% RSLogix 500 project P3_ABIOLA_A.RSS, saved by version 8.30.00.16 %
PROJECT "UNTITLED"    % processor: Bul.1763 MicroLogix 1100 Series B %

PROGRAM FILES
  LAD 2   2 rungs
  LAD 3 "PSEUDO IO"  30 rungs  % Contains all the assigned memery address used  %

DATA FILES
  O0 OUTPUT  4 elements
  I1 INPUT  6 elements
  S2 STATUS  66 elements
  B3 BINARY  1 elements
  T4 TIMER  7 elements
  C5 COUNTER  6 elements
  R6 CONTROL  1 elements
  N7 INTEGER  30 elements
  F8 FLOAT  1 elements
  ST9 STRFRBCSCN  50 elements  % Writes string from bar code scanner to PLC %

LADDER 2
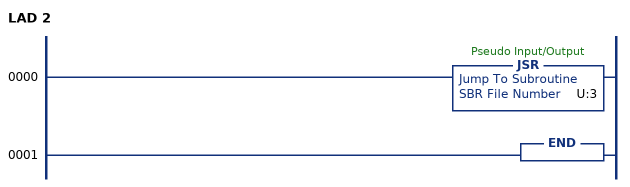
% Rung: 0 %
SOR JSR U:3 EOR
%   U:3  "Pseudo Input/Output" %
% Rung: 1 %
SOR END EOR

LADDER 3 "PSEUDO IO"    % Contains all the assigned memery address used  %
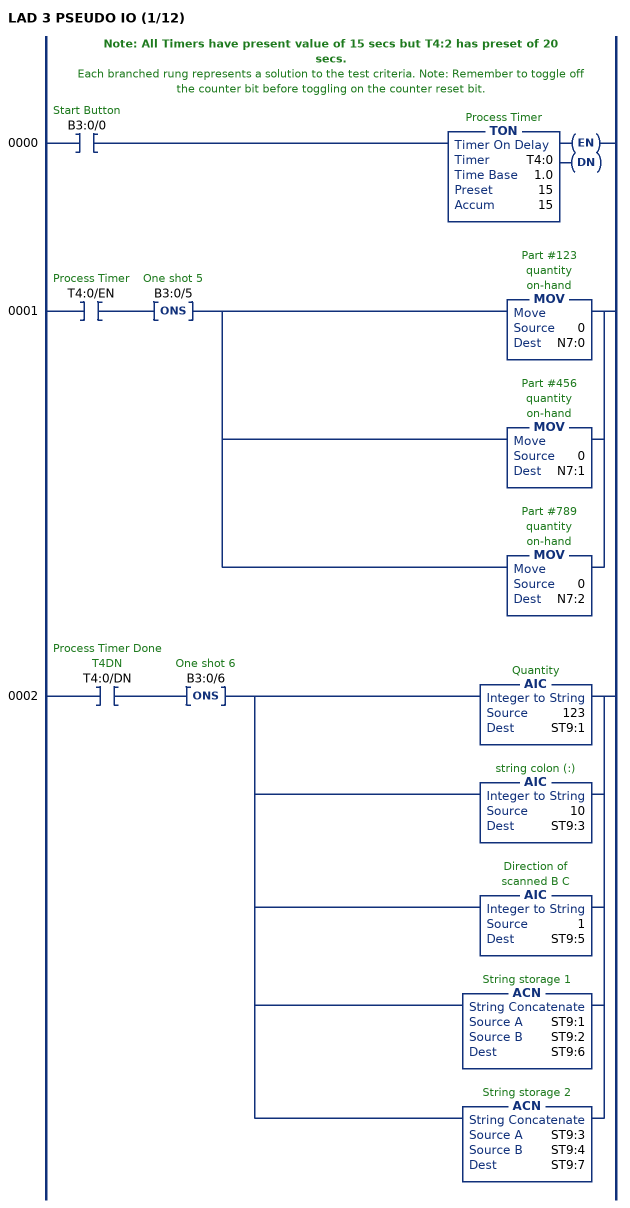
% Rung: 0 %
% TITLE: Note: All Timers have present value of 15 secs but T4:2 has preset of 20 secs. %
% Each branched rung represents a solution to the test criteria. Note: Remember to toggle off the counter bit before toggling on the counter reset bit. %
SOR XIC B3:0/0 TON T4:0 1.0 15 15 EOR
%   B3:0/0  "Start Button" %
%   T4:0  "Process Timer" %
% Rung: 1 %
SOR XIC T4:0/EN ONS B3:0/5 BST MOV 0 N7:0 NXB BST MOV 0 N7:1 NXB MOV 0 N7:2 BND BND EOR
%   T4:0  "Process Timer" %
%   B3:0/5  "One shot 5" %
%   N7:0  "Part #123 quantity on-hand" %
%   N7:1  "Part #456 quantity on-hand" %
%   N7:2  "Part #789 quantity on-hand" %
% Rung: 2 %
SOR XIC T4:0/DN ONS B3:0/6 BST AIC 123 ST9:1 NXB BST AIC 10 ST9:3 NXB BST AIC 1 ST9:5 NXB BST ACN ST9:1 ST9:2 ST9:6 NXB ACN ST9:3 ST9:4 ST9:7 BND BND BND BND EOR
%   T4:0/DN  T4DN  "Process Timer Done" %
%   B3:0/6  "One shot 6" %
%   ST9:1  "Quantity" %
%   ST9:3  "string colon (:)" %
%   ST9:5  "Direction of scanned B C" %
%   ST9:2  "String Quantity from Bar-code scanner" %
%   ST9:6  "String storage 1" %
%   ST9:4  "Concatination of colon (:) with direction from BCS" %
%   ST9:7  "String storage 2" %

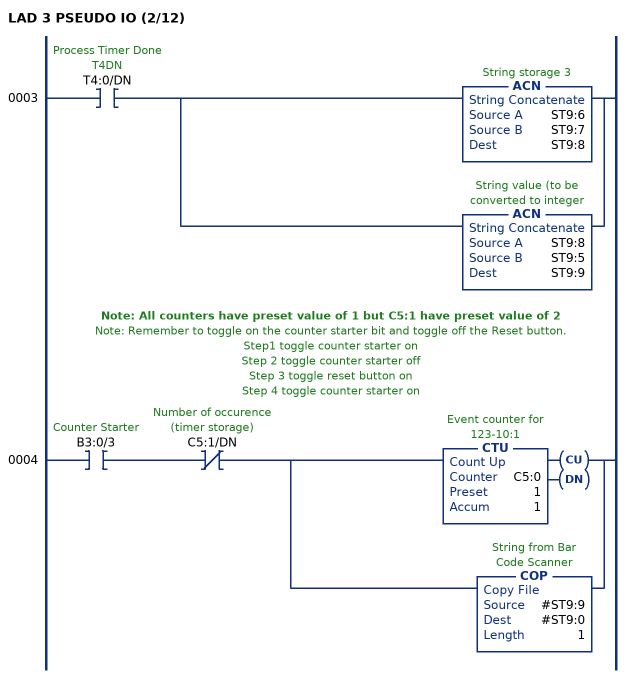
% Rung: 3 %
SOR XIC T4:0/DN BST ACN ST9:6 ST9:7 ST9:8 NXB ACN ST9:8 ST9:5 ST9:9 BND EOR
%   T4:0/DN  T4DN  "Process Timer Done" %
%   ST9:6  "String storage 1" %
%   ST9:7  "String storage 2" %
%   ST9:8  "String storage 3" %
%   ST9:5  "Direction of scanned B C" %
%   ST9:9  "String value (to be converted to integer" %
% Rung: 4 %
% TITLE: Note: All counters have preset value of 1 but C5:1 have preset value of 2 %
% Note: Remember to toggle on the counter starter bit and toggle off the Reset button.
% Step1 toggle counter starter on
% Step 2 toggle counter starter off
% Step 3 toggle reset button on
% Step 4 toggle counter starter on %
SOR XIC B3:0/3 XIO C5:1/DN BST CTU C5:0 1 1 NXB COP #ST9:9 #ST9:0 1 BND EOR
%   B3:0/3  "Counter Starter" %
%   C5:1/DN  "Number of occurence (timer storage)" %
%   C5:0  "Event counter for 123-10:1" %
%   ST9:9  "String value (to be converted to integer" %
%   ST9:0  "String from Bar Code Scanner" %

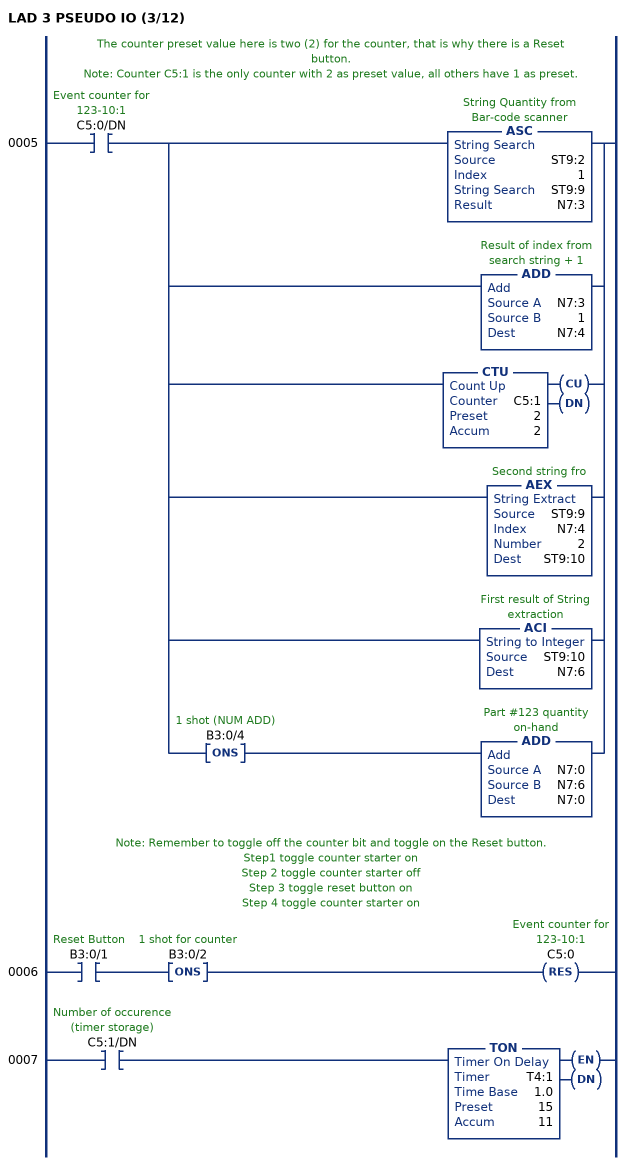
% Rung: 5 %
% The counter preset value here is two (2) for the counter, that is why there is a Reset button.
% Note: Counter C5:1 is the only counter with 2 as preset value, all others have 1 as preset. %
SOR XIC C5:0/DN BST BST ASC ST9:2 1 ST9:9 N7:3 NXB BST ADD N7:3 1 N7:4 NXB CTU C5:1 2 2 BND BND NXB BST AEX ST9:9 N7:4 2 ST9:10 NXB BST ACI ST9:10 N7:6 NXB ONS B3:0/4 ADD N7:0 N7:6 N7:0 BND BND BND EOR
%   C5:0  "Event counter for 123-10:1" %
%   ST9:2  "String Quantity from Bar-code scanner" %
%   ST9:9  "String value (to be converted to integer" %
%   N7:3  "Constant value of 10" %
%   N7:4  "Result of index from search string + 1" %
%   ST9:10  "Second string fro" %
%   N7:6  "First result of String extraction" %
%   B3:0/4  "1 shot (NUM ADD)" %
%   N7:0  "Part #123 quantity on-hand" %
% Rung: 6 %
% Note: Remember to toggle off the counter bit and toggle on the Reset button.
% Step1 toggle counter starter on
% Step 2 toggle counter starter off
% Step 3 toggle reset button on
% Step 4 toggle counter starter on %
SOR XIC B3:0/1 ONS B3:0/2 RES C5:0 EOR
%   B3:0/1  "Reset Button" %
%   B3:0/2  "1 shot for counter" %
%   C5:0  "Event counter for 123-10:1" %
% Rung: 7 %
SOR XIC C5:1/DN TON T4:1 1.0 15 11 EOR
%   C5:1/DN  "Number of occurence (timer storage)" %

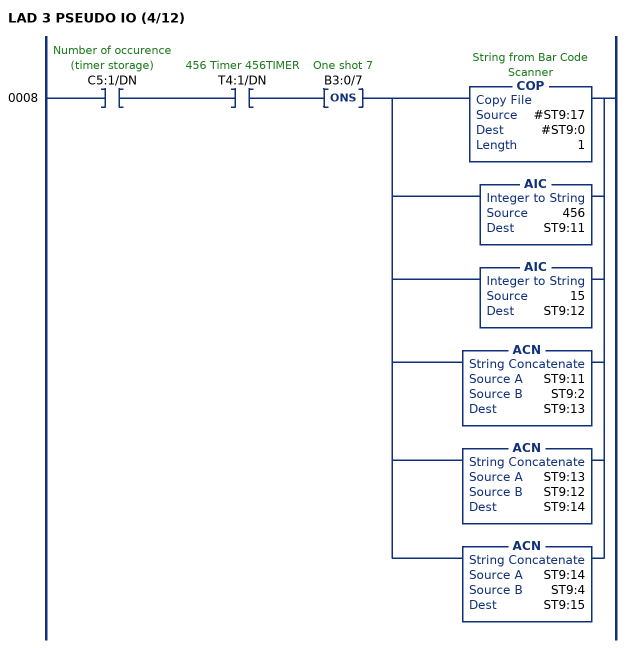
% Rung: 8 %
SOR XIC C5:1/DN XIC T4:1/DN ONS B3:0/7 BST BST COP #ST9:17 #ST9:0 1 NXB AIC 456 ST9:11 BND NXB AIC 15 ST9:12 NXB ACN ST9:11 ST9:2 ST9:13 NXB ACN ST9:13 ST9:12 ST9:14 NXB ACN ST9:14 ST9:4 ST9:15 BND EOR
%   C5:1/DN  "Number of occurence (timer storage)" %
%   T4:1/DN  456TIMER  "456 Timer" %
%   B3:0/7  "One shot 7" %
%   ST9:0  "String from Bar Code Scanner" %
%   ST9:2  "String Quantity from Bar-code scanner" %
%   ST9:4  "Concatination of colon (:) with direction from BCS" %

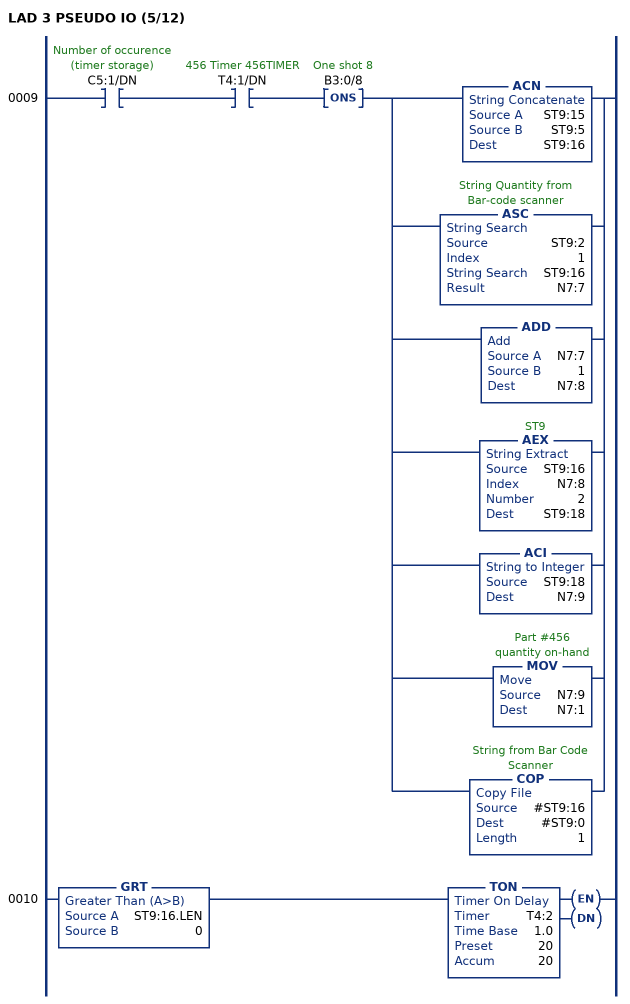
% Rung: 9 %
SOR XIC C5:1/DN XIC T4:1/DN ONS B3:0/8 BST ACN ST9:15 ST9:5 ST9:16 NXB ASC ST9:2 1 ST9:16 N7:7 NXB BST ADD N7:7 1 N7:8 NXB BST BST AEX ST9:16 N7:8 2 ST9:18 NXB ACI ST9:18 N7:9 BND NXB BST MOV N7:9 N7:1 NXB COP #ST9:16 #ST9:0 1 BND BND BND BND EOR
%   C5:1/DN  "Number of occurence (timer storage)" %
%   T4:1/DN  456TIMER  "456 Timer" %
%   B3:0/8  "One shot 8" %
%   ST9:5  "Direction of scanned B C" %
%   ST9:2  "String Quantity from Bar-code scanner" %
%   ST9:18  ST9 %
%   N7:1  "Part #456 quantity on-hand" %
%   ST9:0  "String from Bar Code Scanner" %
% Rung: 10 %
SOR GRT ST9:16.LEN 0 TON T4:2 1.0 20 20 EOR

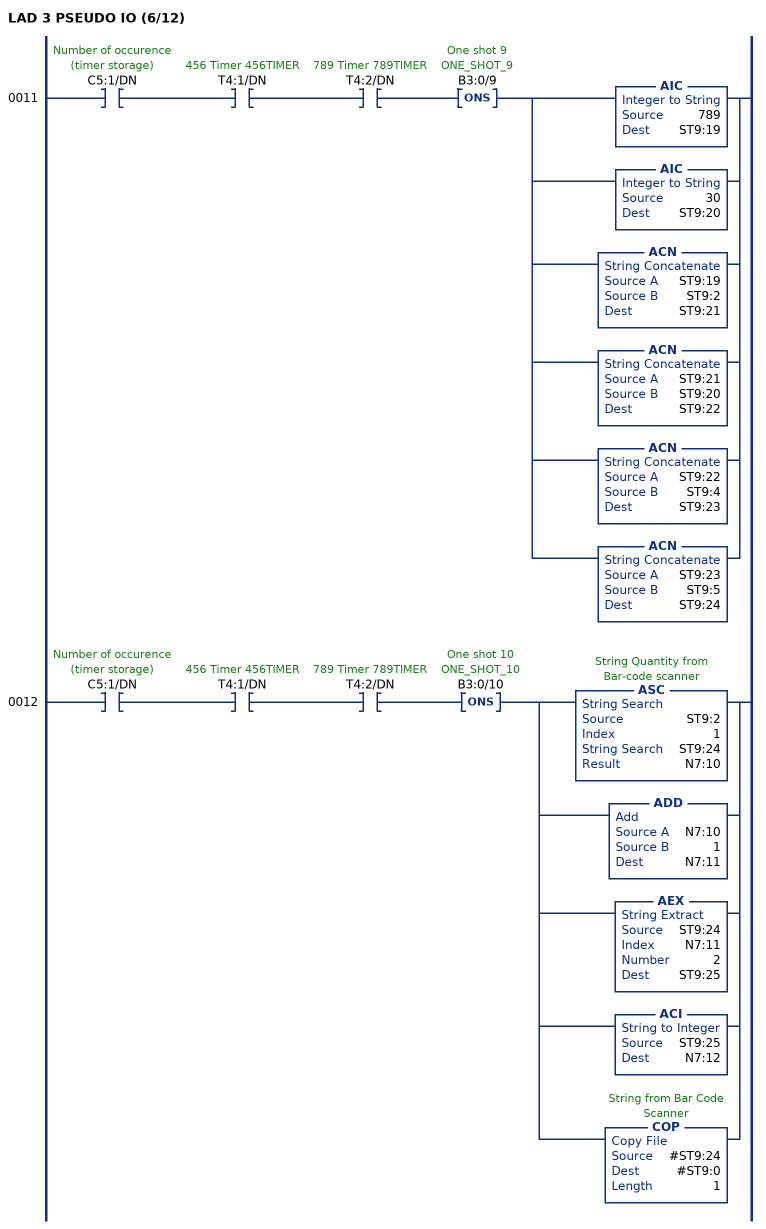
% Rung: 11 %
SOR XIC C5:1/DN XIC T4:1/DN XIC T4:2/DN ONS B3:0/9 BST AIC 789 ST9:19 NXB AIC 30 ST9:20 NXB ACN ST9:19 ST9:2 ST9:21 NXB ACN ST9:21 ST9:20 ST9:22 NXB ACN ST9:22 ST9:4 ST9:23 NXB ACN ST9:23 ST9:5 ST9:24 BND EOR
%   C5:1/DN  "Number of occurence (timer storage)" %
%   T4:1/DN  456TIMER  "456 Timer" %
%   T4:2/DN  789TIMER  "789 Timer" %
%   B3:0/9  ONE_SHOT_9  "One shot 9" %
%   ST9:2  "String Quantity from Bar-code scanner" %
%   ST9:4  "Concatination of colon (:) with direction from BCS" %
%   ST9:5  "Direction of scanned B C" %
% Rung: 12 %
SOR XIC C5:1/DN XIC T4:1/DN XIC T4:2/DN ONS B3:0/10 BST ASC ST9:2 1 ST9:24 N7:10 NXB BST ADD N7:10 1 N7:11 NXB BST AEX ST9:24 N7:11 2 ST9:25 NXB BST ACI ST9:25 N7:12 NXB COP #ST9:24 #ST9:0 1 BND BND BND BND EOR
%   C5:1/DN  "Number of occurence (timer storage)" %
%   T4:1/DN  456TIMER  "456 Timer" %
%   T4:2/DN  789TIMER  "789 Timer" %
%   B3:0/10  ONE_SHOT_10  "One shot 10" %
%   ST9:2  "String Quantity from Bar-code scanner" %
%   ST9:0  "String from Bar Code Scanner" %

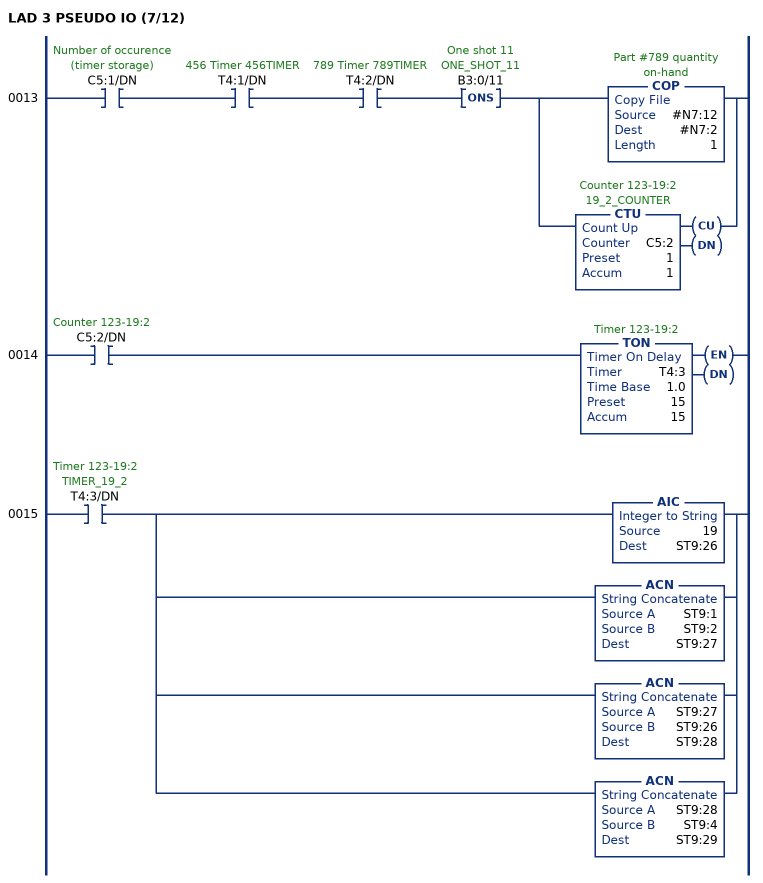
% Rung: 13 %
SOR XIC C5:1/DN XIC T4:1/DN XIC T4:2/DN ONS B3:0/11 BST COP #N7:12 #N7:2 1 NXB CTU C5:2 1 1 BND EOR
%   C5:1/DN  "Number of occurence (timer storage)" %
%   T4:1/DN  456TIMER  "456 Timer" %
%   T4:2/DN  789TIMER  "789 Timer" %
%   B3:0/11  ONE_SHOT_11  "One shot 11" %
%   N7:2  "Part #789 quantity on-hand" %
%   C5:2  19_2_COUNTER  "Counter 123-19:2" %
% Rung: 14 %
SOR XIC C5:2/DN TON T4:3 1.0 15 15 EOR
%   C5:2/DN  "Counter 123-19:2" %
%   T4:3  "Timer 123-19:2" %
% Rung: 15 %
SOR XIC T4:3/DN BST AIC 19 ST9:26 NXB BST ACN ST9:1 ST9:2 ST9:27 NXB BST ACN ST9:27 ST9:26 ST9:28 NXB ACN ST9:28 ST9:4 ST9:29 BND BND BND EOR
%   T4:3/DN  TIMER_19_2  "Timer 123-19:2" %
%   ST9:1  "Quantity" %
%   ST9:2  "String Quantity from Bar-code scanner" %
%   ST9:4  "Concatination of colon (:) with direction from BCS" %

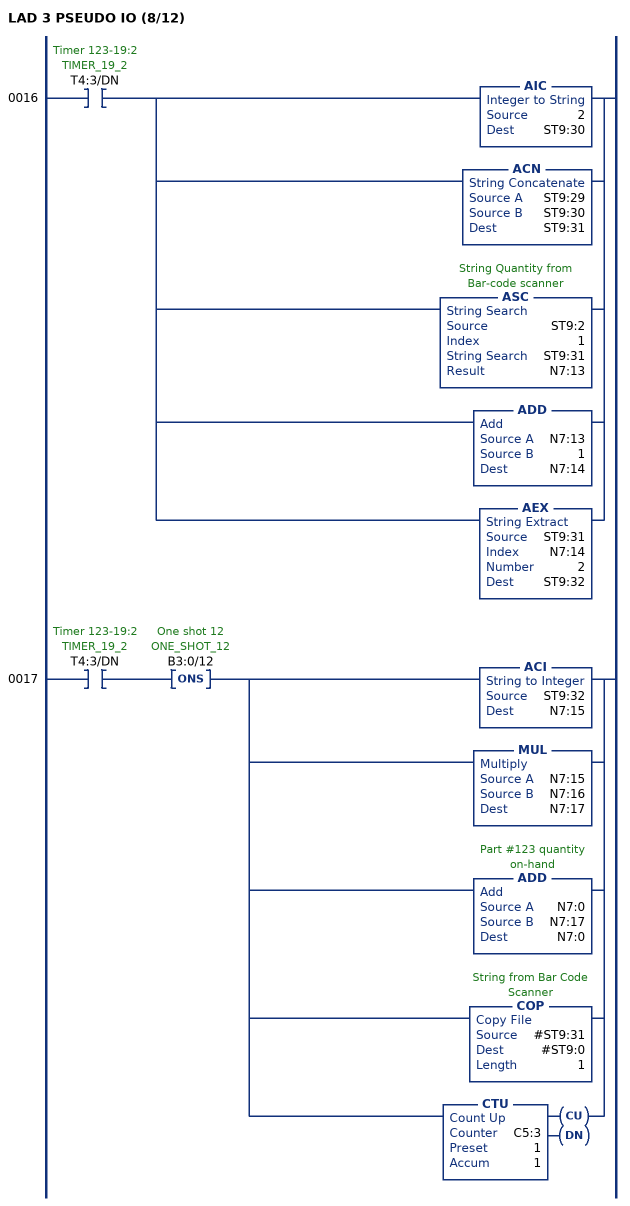
% Rung: 16 %
SOR XIC T4:3/DN BST AIC 2 ST9:30 NXB BST ACN ST9:29 ST9:30 ST9:31 NXB BST ASC ST9:2 1 ST9:31 N7:13 NXB BST ADD N7:13 1 N7:14 NXB AEX ST9:31 N7:14 2 ST9:32 BND BND BND BND EOR
%   T4:3/DN  TIMER_19_2  "Timer 123-19:2" %
%   ST9:2  "String Quantity from Bar-code scanner" %
% Rung: 17 %
SOR XIC T4:3/DN ONS B3:0/12 BST BST ACI ST9:32 N7:15 NXB MUL N7:15 N7:16 N7:17 BND NXB BST ADD N7:0 N7:17 N7:0 NXB BST COP #ST9:31 #ST9:0 1 NXB CTU C5:3 1 1 BND BND BND EOR
%   T4:3/DN  TIMER_19_2  "Timer 123-19:2" %
%   B3:0/12  ONE_SHOT_12  "One shot 12" %
%   N7:16  N %
%   N7:0  "Part #123 quantity on-hand" %
%   ST9:0  "String from Bar Code Scanner" %

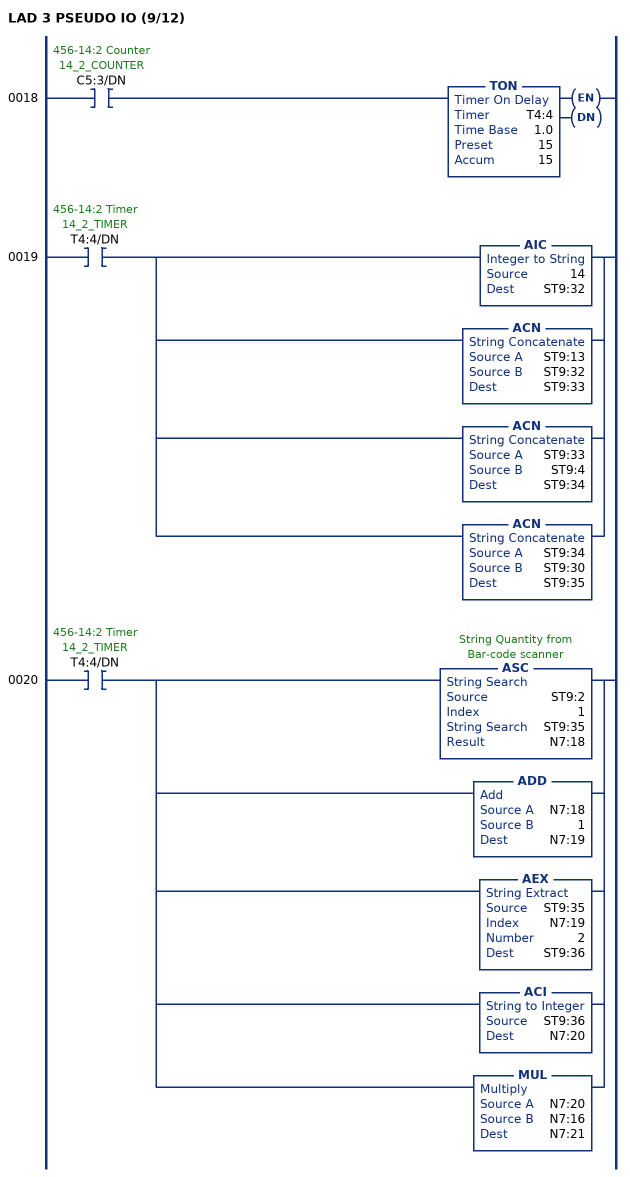
% Rung: 18 %
SOR XIC C5:3/DN TON T4:4 1.0 15 15 EOR
%   C5:3/DN  14_2_COUNTER  "456-14:2 Counter" %
% Rung: 19 %
SOR XIC T4:4/DN BST AIC 14 ST9:32 NXB BST ACN ST9:13 ST9:32 ST9:33 NXB BST ACN ST9:33 ST9:4 ST9:34 NXB ACN ST9:34 ST9:30 ST9:35 BND BND BND EOR
%   T4:4/DN  14_2_TIMER  "456-14:2 Timer" %
%   ST9:4  "Concatination of colon (:) with direction from BCS" %
% Rung: 20 %
SOR XIC T4:4/DN BST ASC ST9:2 1 ST9:35 N7:18 NXB BST ADD N7:18 1 N7:19 NXB BST AEX ST9:35 N7:19 2 ST9:36 NXB BST ACI ST9:36 N7:20 NXB MUL N7:20 N7:16 N7:21 BND BND BND BND EOR
%   T4:4/DN  14_2_TIMER  "456-14:2 Timer" %
%   ST9:2  "String Quantity from Bar-code scanner" %
%   N7:16  N %

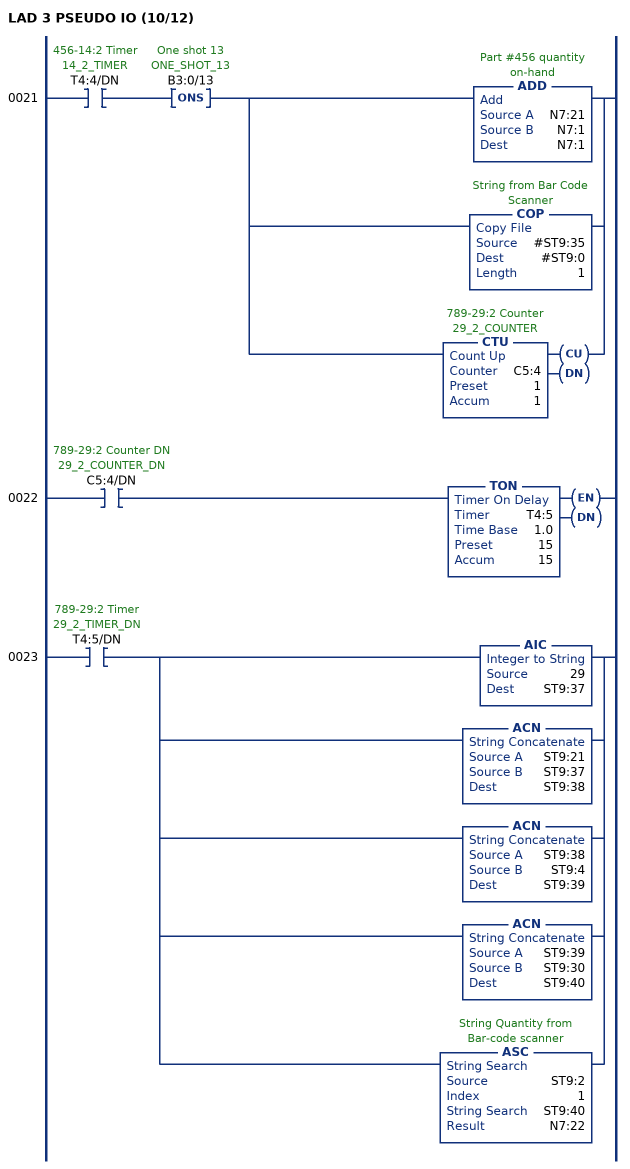
% Rung: 21 %
SOR XIC T4:4/DN ONS B3:0/13 BST ADD N7:21 N7:1 N7:1 NXB BST COP #ST9:35 #ST9:0 1 NXB CTU C5:4 1 1 BND BND EOR
%   T4:4/DN  14_2_TIMER  "456-14:2 Timer" %
%   B3:0/13  ONE_SHOT_13  "One shot 13" %
%   N7:1  "Part #456 quantity on-hand" %
%   ST9:0  "String from Bar Code Scanner" %
%   C5:4  29_2_COUNTER  "789-29:2 Counter" %
% Rung: 22 %
SOR XIC C5:4/DN TON T4:5 1.0 15 15 EOR
%   C5:4/DN  29_2_COUNTER_DN  "789-29:2 Counter DN" %
% Rung: 23 %
SOR XIC T4:5/DN BST AIC 29 ST9:37 NXB BST ACN ST9:21 ST9:37 ST9:38 NXB BST ACN ST9:38 ST9:4 ST9:39 NXB BST ACN ST9:39 ST9:30 ST9:40 NXB ASC ST9:2 1 ST9:40 N7:22 BND BND BND BND EOR
%   T4:5/DN  29_2_TIMER_DN  "789-29:2 Timer" %
%   ST9:4  "Concatination of colon (:) with direction from BCS" %
%   ST9:2  "String Quantity from Bar-code scanner" %

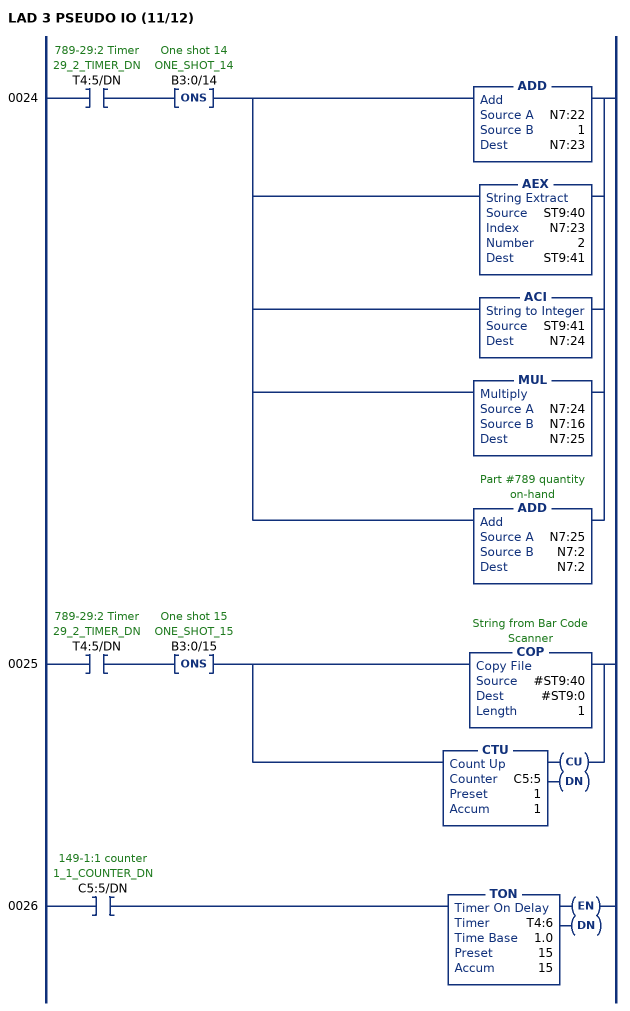
% Rung: 24 %
SOR XIC T4:5/DN ONS B3:0/14 BST ADD N7:22 1 N7:23 NXB BST AEX ST9:40 N7:23 2 ST9:41 NXB BST ACI ST9:41 N7:24 NXB MUL N7:24 N7:16 N7:25 NXB ADD N7:25 N7:2 N7:2 BND BND BND EOR
%   T4:5/DN  29_2_TIMER_DN  "789-29:2 Timer" %
%   B3:0/14  ONE_SHOT_14  "One shot 14" %
%   N7:16  N %
%   N7:2  "Part #789 quantity on-hand" %
% Rung: 25 %
SOR XIC T4:5/DN ONS B3:0/15 BST COP #ST9:40 #ST9:0 1 NXB CTU C5:5 1 1 BND EOR
%   T4:5/DN  29_2_TIMER_DN  "789-29:2 Timer" %
%   B3:0/15  ONE_SHOT_15  "One shot 15" %
%   ST9:0  "String from Bar Code Scanner" %
% Rung: 26 %
SOR XIC C5:5/DN TON T4:6 1.0 15 15 EOR
%   C5:5/DN  1_1_COUNTER_DN  "149-1:1 counter" %

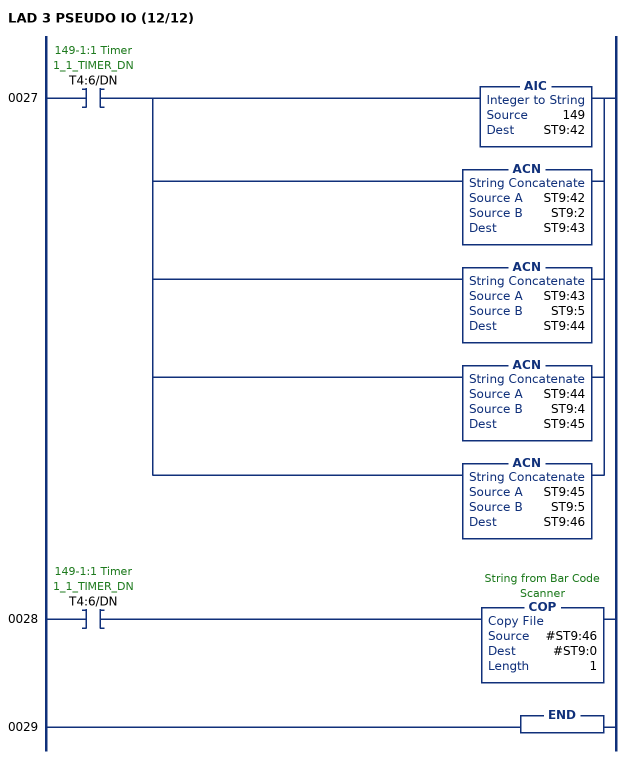
% Rung: 27 %
SOR XIC T4:6/DN BST AIC 149 ST9:42 NXB BST ACN ST9:42 ST9:2 ST9:43 NXB BST ACN ST9:43 ST9:5 ST9:44 NXB BST ACN ST9:44 ST9:4 ST9:45 NXB ACN ST9:45 ST9:5 ST9:46 BND BND BND BND EOR
%   T4:6/DN  1_1_TIMER_DN  "149-1:1 Timer" %
%   ST9:2  "String Quantity from Bar-code scanner" %
%   ST9:5  "Direction of scanned B C" %
%   ST9:4  "Concatination of colon (:) with direction from BCS" %
% Rung: 28 %
SOR XIC T4:6/DN COP #ST9:46 #ST9:0 1 EOR
%   T4:6/DN  1_1_TIMER_DN  "149-1:1 Timer" %
%   ST9:0  "String from Bar Code Scanner" %
% Rung: 29 %
SOR END EOR

OTHER DOCUMENTED ADDRESSES
  C5:0.ACC  "Number of count storage"
  C5:0/CU  "Process counter"
  N7:5  "String colon (:) converted to integer"
  ST9:2.0  "Result of Constant Multiplication with -1"
  ST10:1.0  "String len"

DATA TABLE (non-zero values as saved)
DATA B3
% B3:0 % 0X007F
DATA T4
% .PRE .ACC %
% T4:0 % 15 15
% T4:1 % 15 13
% T4:2 % 20 20
% T4:3 % 15 15
% T4:4 % 15 15
% T4:5 % 15 15
% T4:6 % 15 15
DATA C5
% .PRE .ACC %
% C5:0 % 1 1
% C5:1 % 2 2
% C5:2 % 1 1
% C5:3 % 1 1
% C5:4 % 1 1
% C5:5 % 1 1
DATA N7
% N7:0 % 1 1 1 4 5 0 10 4 5 15
% N7:10 % 4 5 30 4 5 19 -1 -19 4 5
% N7:20 % 14 -14 4 5 29 -29 0 0 0 0
DATA ST9
% ST9:0 % "149-1:1"
% ST9:1 % "123"
% ST9:2 % "-"
% ST9:3 % "10"
% ST9:4 % ":"
% ST9:5 % "1"
% ST9:6 % "123-"
% ST9:7 % "10:"
% ST9:8 % "123-10:"
% ST9:9 % "123-10:1"
% ST9:10 % "10"
% ST9:11 % "456"
% ST9:12 % "15"
% ST9:13 % "456-"
% ST9:14 % "456-15"
% ST9:15 % "456-15:"
% ST9:16 % "456-15:1"
% ST9:17 % " "
% ST9:18 % "15"
% ST9:19 % "789"
% ST9:20 % "30"
% ST9:21 % "789-"
% ST9:22 % "789-30"
% ST9:23 % "789-30:"
% ST9:24 % "789-30:1"
% ST9:25 % "30"
% ST9:26 % "19"
% ST9:27 % "123-"
% ST9:28 % "123-19"
% ST9:29 % "123-19:"
% ST9:30 % "2"
% ST9:31 % "123-19:2"
% ST9:32 % "14"
% ST9:33 % "456-14"
% ST9:34 % "456-14:"
% ST9:35 % "456-14:2"
% ST9:36 % "14"
% ST9:37 % "29"
% ST9:38 % "789-29"
% ST9:39 % "789-29:"
% ST9:40 % "789-29:2"
% ST9:41 % "29"
% ST9:42 % "149"
% ST9:43 % "149-"
% ST9:44 % "149-1"
% ST9:45 % "149-1:"
% ST9:46 % "149-1:1"
